Staubli VAL3: BuildFrame.pgx

public program BuildFrame(string x_sFrameName, frame& x_fFrame[], num& x_nError[])
  local num l_nRadius
  local trsf l_tfCenter
  local point l_pCenter
begin
  // This program calculates the conveyor reference frame
  // depending on the type of conveyor (linear or circular)
  //
  // Input Param
  //
  //
  // Output Param
  // x_fCOnveyor   : reference frame of conveyor
  //
  // Miscellaneous
  //
  // Created 23-02-05                                   C.CURRIVAND
  //----------------------------------------------------------------
  //
  if x_sFrameName=="conveyor"
    if bLinear
      x_nError=setFrame(pWinUp[0],pWinDown[0],pWinUp[1],x_fFrame)
    else
      call ut:centerCircle(pWinUp[0],pWinMiddle,pWinDown[0],l_tfCenter,l_nRadius)
      l_pCenter=pWinUp[0]
      l_pCenter.trsf=l_tfCenter
      x_nError=setFrame(l_pCenter,pWinUp[0],pWinDown[0],x_fFrame)
    endIf
  else
    x_nError=setFrame(pVision[0],pVision[1],pVision[2],x_fFrame)
  endIf
end
